// TIA Portal V15.1 export
// export: Created 2020-06-12T07:35:54.1162109Z, ExportSetting None, DisplayName Totally Integrated Automation Portal, DisplayVersion V15.1, DisplayName TIA Portal Openness, DisplayVersion V15.1, DisplayName STEP 7 Professional, DisplayVersion V15.1, DisplayName STEP 7 Safety, DisplayVersion V15.1, DisplayName WinCC Advanced, DisplayVersion V15.1
FUNCTION "RCW_call" : Void   // FC182, FBD
{ S7_Optimized_Access := 'TRUE' }
// stored: SetENOAutomatically False
BEGIN

REGION Network 1: Pumps logic
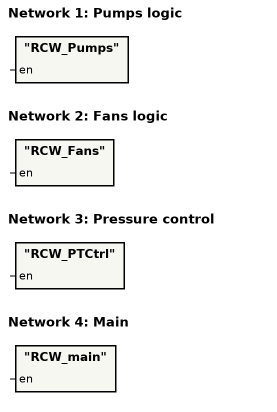
   "RCW_Pumps"();
END_REGION

REGION Network 2: Fans logic
   "RCW_Fans"();
END_REGION

REGION Network 3: Pressure control
   "RCW_PTCtrl"();
END_REGION

REGION Network 4: Main
   "RCW_main"();
END_REGION
END_FUNCTION
